Yaskawa INFORM job: ARGAZ_PROGRAM.JBI

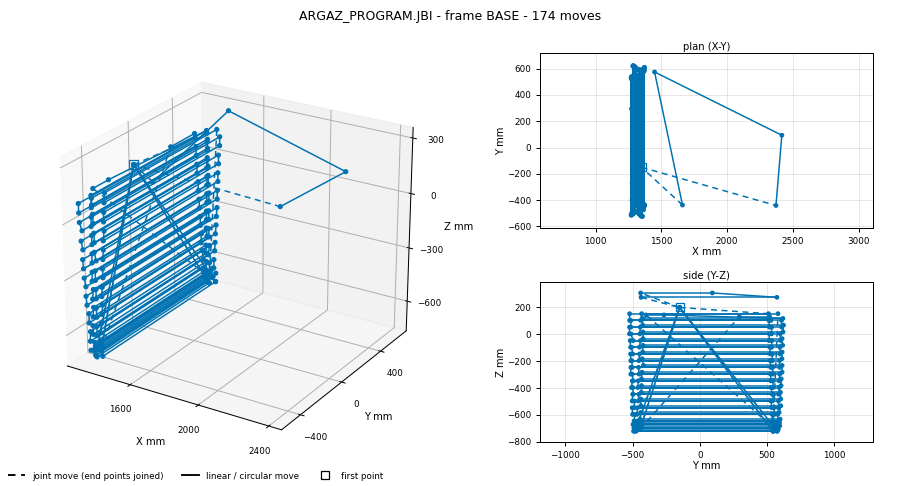
[picture p0: tool path of ARGAZ_PROGRAM.JBI in frame BASE, 174 of 174 moves have a stored position in this frame; points joined in program order, loops and branches not executed]
/JOB
//NAME ARGAZ_PROGRAM
//POS
///NPOS 168,0,168,1,0,1
///TOOL 0
///POSTYPE BASE
///RECTAN
///RCONF 0,0,0,0,0,0,0,0,0,0,0,0,0,0,0,0,0,0,0,0,0,0,0,0
C00000=2371.989,-440.401,308.020,175.0000,5.0000,90.0000
C00001=2416.705,93.738,308.020,175.0000,5.0000,90.0000
C00002=1448.862,574.607,275.381,175.0000,5.0000,90.0000
C00003=1661.240,-437.144,275.381,175.0000,5.0000,90.0000
C00004=1357.088,511.287,153.366,175.0000,-89.9999,5.0000
C00005=1357.088,-522.394,153.366,175.0000,-89.9999,5.0000
C00006=1354.164,-522.287,103.366,175.0000,-89.9999,5.0000
C00007=1354.164,514.938,103.366,175.0000,-89.9999,5.0000
C00008=1352.438,518.625,53.366,175.0000,-89.9999,5.0000
C00009=1352.438,-522.994,53.366,175.0000,-89.9999,5.0000
C00010=1350.832,-523.178,3.366,175.0000,-89.9999,5.0000
C00011=1350.832,518.871,3.366,175.0000,-89.9999,5.0000
C00012=1348.825,516.219,-46.633,175.0000,-89.9999,5.0000
C00013=1348.825,-518.107,-46.633,175.0000,-89.9999,5.0000
C00014=1347.044,-514.870,-96.633,175.0000,-89.9999,5.0000
C00015=1347.044,522.164,-96.633,175.0000,-89.9999,5.0000
C00016=1345.183,525.111,-146.633,175.0000,-89.9999,5.0000
C00017=1345.183,-515.018,-146.633,175.0000,-89.9999,5.0000
C00018=1343.293,-513.493,-196.633,175.0000,-89.9999,5.0000
C00019=1343.293,525.184,-196.633,175.0000,-89.9999,5.0000
C00020=1341.807,528.689,-246.633,175.0000,-89.9999,5.0000
C00021=1341.807,-512.923,-246.633,175.0000,-89.9999,5.0000
C00022=1339.870,-513.256,-296.633,175.0000,-89.9999,5.0000
C00023=1339.870,527.209,-296.633,175.0000,-89.9999,5.0000
C00024=1337.995,529.873,-346.633,175.0000,-89.9999,5.0000
C00025=1337.995,-502.334,-346.633,175.0000,-89.9999,5.0000
C00026=1336.213,-508.248,-396.633,175.0000,-89.9999,5.0000
C00027=1336.213,530.626,-396.633,175.0000,-89.9999,5.0000
C00028=1334.396,540.131,-446.633,175.0000,-89.9999,5.0000
C00029=1334.396,-499.231,-446.633,175.0000,-89.9999,5.0000
C00030=1332.129,-503.451,-496.633,175.0000,-89.9999,5.0000
C00031=1332.129,530.722,-496.633,175.0000,-89.9999,5.0000
C00032=1330.170,536.350,-546.633,175.0000,-89.9999,5.0000
C00033=1330.170,-503.270,-546.633,175.0000,-89.9999,5.0000
C00034=1328.250,-500.170,-596.633,175.0000,-89.9999,5.0000
C00035=1328.250,538.973,-596.633,175.0000,-89.9999,5.0000
C00036=1326.642,540.301,-646.633,175.0000,-89.9999,5.0000
C00037=1326.642,-487.964,-646.633,175.0000,-89.9999,5.0000
C00038=1324.806,-489.352,-696.633,175.0000,-89.9999,5.0000
C00039=1324.806,541.085,-696.633,175.0000,-89.9999,5.0000
C00040=1343.412,545.195,-671.633,180.0000,-60.0000,0.0000
C00041=1343.412,-497.251,-671.633,180.0000,-60.0000,0.0000
C00042=1342.156,-493.079,-721.633,180.0000,-60.0000,0.0000
C00043=1342.156,545.345,-721.633,180.0000,-60.0000,0.0000
C00044=1342.156,545.345,-721.633,180.0000,-60.0000,0.0000
C00045=1371.377,582.641,153.649,175.0000,-89.9999,5.0000
C00046=1371.377,-432.613,153.649,175.0000,-89.9999,5.0000
C00047=1372.180,-440.408,103.649,175.0000,-89.9999,5.0000
C00048=1372.180,609.123,103.649,175.0000,-89.9999,5.0000
C00049=1371.089,609.796,53.649,175.0000,-89.9999,5.0000
C00050=1371.089,-443.667,53.649,175.0000,-89.9999,5.0000
C00051=1369.998,-445.573,3.649,175.0000,-89.9999,5.0000
C00052=1369.998,599.394,3.649,175.0000,-89.9999,5.0000
C00053=1369.110,601.830,-46.350,175.0000,-89.9999,5.0000
C00054=1369.110,-441.873,-46.350,175.0000,-89.9999,5.0000
C00055=1367.639,-448.976,-96.350,175.0000,-89.9999,5.0000
C00056=1367.639,596.630,-96.350,175.0000,-89.9999,5.0000
C00057=1366.582,598.500,-146.350,175.0000,-89.9999,5.0000
C00058=1366.582,-448.746,-146.350,175.0000,-89.9999,5.0000
C00059=1365.085,-453.213,-196.350,175.0000,-89.9999,5.0000
C00060=1365.085,594.650,-196.350,175.0000,-89.9999,5.0000
C00061=1363.658,594.990,-246.350,175.0000,-89.9999,5.0000
C00062=1363.658,-455.754,-246.350,175.0000,-89.9999,5.0000
C00063=1361.864,-451.909,-296.350,175.0000,-89.9999,5.0000
C00064=1361.864,595.571,-296.350,175.0000,-89.9999,5.0000
C00065=1360.073,591.872,-346.350,175.0000,-89.9999,5.0000
C00066=1360.073,-458.655,-346.350,175.0000,-89.9999,5.0000
C00067=1358.161,-460.748,-396.350,175.0000,-89.9999,5.0000
C00068=1358.161,591.928,-396.350,175.0000,-89.9999,5.0000
C00069=1356.405,587.009,-446.350,175.0000,-89.9999,5.0000
C00070=1356.405,-453.709,-446.350,175.0000,-89.9999,5.0000
C00071=1354.608,-458.341,-496.350,175.0000,-89.9999,5.0000
C00072=1354.608,586.376,-496.350,175.0000,-89.9999,5.0000
C00073=1352.468,585.807,-546.350,175.0000,-89.9999,5.0000
C00074=1352.468,-463.981,-546.350,175.0000,-89.9999,5.0000
C00075=1350.405,-467.600,-596.350,175.0000,-89.9999,5.0000
C00076=1350.405,580.519,-596.350,175.0000,-89.9999,5.0000
C00077=1348.479,582.258,-646.350,175.0000,-89.9999,5.0000
C00078=1348.479,-467.412,-646.350,175.0000,-89.9999,5.0000
C00079=1346.462,-469.588,-696.350,175.0000,-89.9999,5.0000
C00080=1346.462,577.739,-696.350,175.0000,-89.9999,5.0000
C00081=1364.869,576.218,-671.350,180.0000,-60.0000,0.0000
C00082=1364.869,-472.867,-671.350,180.0000,-60.0000,0.0000
C00083=1363.104,-472.908,-721.350,180.0000,-60.0000,0.0000
C00084=1363.104,576.344,-721.350,180.0000,-60.0000,0.0000
C00085=1363.104,576.344,-721.350,180.0000,-60.0000,0.0000
C00086=1277.888,-399.618,144.199,175.0000,-89.9999,5.0000
C00087=1277.888,-266.558,144.199,175.0000,-89.9999,5.0000
C00088=1283.410,619.398,117.816,175.0000,-89.9999,5.0000
C00089=1283.410,-424.812,117.816,175.0000,-89.9999,5.0000
C00090=1286.253,-425.480,67.816,175.0000,-89.9999,5.0000
C00091=1286.253,623.737,67.816,175.0000,-89.9999,5.0000
C00092=1288.733,620.101,17.816,175.0000,-89.9999,5.0000
C00093=1288.733,-423.231,17.816,175.0000,-89.9999,5.0000
C00094=1291.050,-422.345,-32.183,175.0000,-89.9999,5.0000
C00095=1291.050,613.233,-32.183,175.0000,-89.9999,5.0000
C00096=1293.592,617.319,-82.183,175.0000,-89.9999,5.0000
C00097=1293.592,-423.386,-82.183,175.0000,-89.9999,5.0000
C00098=1295.614,-424.881,-132.183,175.0000,-89.9999,5.0000
C00099=1295.614,613.520,-132.183,175.0000,-89.9999,5.0000
C00100=1297.247,612.008,-182.183,175.0000,-89.9999,5.0000
C00101=1297.247,-429.228,-182.183,175.0000,-89.9999,5.0000
C00102=1299.433,-419.216,-232.183,175.0000,-89.9999,5.0000
C00103=1299.433,613.471,-232.183,175.0000,-89.9999,5.0000
C00104=1300.418,613.420,-282.183,175.0000,-89.9999,5.0000
C00105=1300.418,-430.256,-282.183,175.0000,-89.9999,5.0000
C00106=1302.234,-433.734,-332.183,175.0000,-89.9999,5.0000
C00107=1302.234,606.925,-332.183,175.0000,-89.9999,5.0000
C00108=1303.707,605.868,-382.183,175.0000,-89.9999,5.0000
C00109=1303.707,-433.869,-382.183,175.0000,-89.9999,5.0000
C00110=1305.086,-435.019,-432.183,175.0000,-89.9999,5.0000
C00111=1305.086,600.756,-432.183,175.0000,-89.9999,5.0000
C00112=1306.071,603.429,-482.183,175.0000,-89.9999,5.0000
C00113=1306.071,-438.802,-482.183,175.0000,-89.9999,5.0000
C00114=1307.412,-438.117,-532.183,175.0000,-89.9999,5.0000
C00115=1307.412,603.875,-532.183,175.0000,-89.9999,5.0000
C00116=1308.466,591.089,-582.183,175.0000,-89.9999,5.0000
C00117=1308.466,-439.996,-582.183,175.0000,-89.9999,5.0000
C00118=1310.304,-445.204,-632.183,175.0000,-89.9999,5.0000
C00119=1310.304,598.888,-632.183,175.0000,-89.9999,5.0000
C00120=1311.312,595.813,-682.183,175.0000,-89.9999,5.0000
C00121=1311.312,-443.494,-682.183,175.0000,-89.9999,5.0000
C00122=1332.658,-435.818,-657.183,180.0000,-60.0000,0.0000
C00123=1332.658,594.168,-657.183,180.0000,-60.0000,0.0000
C00124=1333.118,585.110,-707.183,180.0000,-60.0000,0.0000
C00125=1333.118,-444.618,-707.183,180.0000,-60.0000,0.0000
C00126=1333.118,-444.618,-707.183,180.0000,-60.0000,0.0000
C00127=1273.288,295.502,131.277,175.0000,-89.9999,5.0000
C00128=1273.288,520.035,131.277,175.0000,-89.9999,5.0000
C00129=1270.890,529.755,103.296,175.0000,-89.9999,5.0000
C00130=1270.890,-513.266,103.296,175.0000,-89.9999,5.0000
C00131=1271.533,-513.209,53.296,175.0000,-89.9999,5.0000
C00132=1271.533,535.502,53.296,175.0000,-89.9999,5.0000
C00133=1273.366,534.257,3.296,175.0000,-89.9999,5.0000
C00134=1273.366,-513.096,3.296,175.0000,-89.9999,5.0000
C00135=1275.404,-495.948,-46.703,175.0000,-89.9999,5.0000
C00136=1275.404,536.502,-46.703,175.0000,-89.9999,5.0000
C00137=1277.028,534.815,-96.703,175.0000,-89.9999,5.0000
C00138=1277.028,-508.386,-96.703,175.0000,-89.9999,5.0000
C00139=1279.183,-498.977,-146.703,175.0000,-89.9999,5.0000
C00140=1279.183,540.662,-146.703,175.0000,-89.9999,5.0000
C00141=1280.966,539.787,-196.703,175.0000,-89.9999,5.0000
C00142=1280.966,-505.503,-196.703,175.0000,-89.9999,5.0000
C00143=1282.925,-503.396,-246.703,175.0000,-89.9999,5.0000
C00144=1282.925,542.645,-246.703,175.0000,-89.9999,5.0000
C00145=1285.047,543.565,-296.703,175.0000,-89.9999,5.0000
C00146=1285.047,-503.499,-296.703,175.0000,-89.9999,5.0000
C00147=1287.369,-494.427,-346.703,175.0000,-89.9999,5.0000
C00148=1287.369,546.345,-346.703,175.0000,-89.9999,5.0000
C00149=1289.521,543.757,-396.703,175.0000,-89.9999,5.0000
C00150=1289.521,-498.930,-396.703,175.0000,-89.9999,5.0000
C00151=1291.635,-495.764,-446.703,175.0000,-89.9999,5.0000
C00152=1291.635,549.175,-446.703,175.0000,-89.9999,5.0000
C00153=1293.849,541.736,-496.703,175.0000,-89.9999,5.0000
C00154=1293.849,-485.793,-496.703,175.0000,-89.9999,5.0000
C00155=1295.977,-487.912,-546.703,175.0000,-89.9999,5.0000
C00156=1295.977,552.744,-546.703,175.0000,-89.9999,5.0000
C00157=1298.303,555.349,-596.703,175.0000,-89.9999,5.0000
C00158=1298.303,-482.618,-596.703,175.0000,-89.9999,5.0000
C00159=1300.270,-489.107,-646.703,175.0000,-89.9999,5.0000
C00160=1300.270,549.567,-646.703,175.0000,-89.9999,5.0000
C00161=1302.656,551.655,-696.703,175.0000,-89.9999,5.0000
C00162=1302.656,-488.761,-696.703,175.0000,-89.9999,5.0000
C00163=1324.870,-481.376,-671.703,180.0000,-60.0000,0.0000
C00164=1324.870,551.349,-671.703,180.0000,-60.0000,0.0000
C00165=1327.105,551.261,-721.703,180.0000,-60.0000,0.0000
C00166=1327.105,-481.969,-721.703,180.0000,-60.0000,0.0000
C00167=1327.105,-481.969,-721.703,180.0000,-60.0000,0.0000
///POSTYPE PULSE
///PULSE
EC00000=0
EC00001=0
EC00002=0
EC00003=0
EC00004=0
EC00005=0
EC00006=0
EC00007=0
EC00008=0
EC00009=0
EC00010=0
EC00011=0
EC00012=0
EC00013=0
EC00014=0
EC00015=0
EC00016=0
EC00017=0
EC00018=0
EC00019=0
EC00020=0
EC00021=0
EC00022=0
EC00023=0
EC00024=0
EC00025=0
EC00026=0
EC00027=0
EC00028=0
EC00029=0
EC00030=0
EC00031=0
EC00032=0
EC00033=0
EC00034=0
EC00035=0
EC00036=0
EC00037=0
EC00038=0
EC00039=0
EC00040=0
EC00041=0
EC00042=0
EC00043=0
EC00044=92160
EC00045=92160
EC00046=92160
EC00047=92160
EC00048=92160
EC00049=92160
EC00050=92160
EC00051=92160
EC00052=92160
EC00053=92160
EC00054=92160
EC00055=92160
EC00056=92160
EC00057=92160
EC00058=92160
EC00059=92160
EC00060=92160
EC00061=92160
EC00062=92160
EC00063=92160
EC00064=92160
EC00065=92160
EC00066=92160
EC00067=92160
EC00068=92160
EC00069=92160
EC00070=92160
EC00071=92160
EC00072=92160
EC00073=92160
EC00074=92160
EC00075=92160
EC00076=92160
EC00077=92160
EC00078=92160
EC00079=92160
EC00080=92160
EC00081=92160
EC00082=92160
EC00083=92160
EC00084=92160
EC00085=184320
EC00086=184320
EC00087=184320
EC00088=184320
EC00089=184320
EC00090=184320
EC00091=184320
EC00092=184320
EC00093=184320
EC00094=184320
EC00095=184320
EC00096=184320
EC00097=184320
EC00098=184320
EC00099=184320
EC00100=184320
EC00101=184320
EC00102=184320
EC00103=184320
EC00104=184320
EC00105=184320
EC00106=184320
EC00107=184320
EC00108=184320
EC00109=184320
EC00110=184320
EC00111=184320
EC00112=184320
EC00113=184320
EC00114=184320
EC00115=184320
EC00116=184320
EC00117=184320
EC00118=184320
EC00119=184320
EC00120=184320
EC00121=184320
EC00122=184320
EC00123=184320
EC00124=184320
EC00125=184320
EC00126=276480
EC00127=276480
EC00128=276480
EC00129=276480
EC00130=276480
EC00131=276480
EC00132=276480
EC00133=276480
EC00134=276480
EC00135=276480
EC00136=276480
EC00137=276480
EC00138=276480
EC00139=276480
EC00140=276480
EC00141=276480
EC00142=276480
EC00143=276480
EC00144=276480
EC00145=276480
EC00146=276480
EC00147=276480
EC00148=276480
EC00149=276480
EC00150=276480
EC00151=276480
EC00152=276480
EC00153=276480
EC00154=276480
EC00155=276480
EC00156=276480
EC00157=276480
EC00158=276480
EC00159=276480
EC00160=276480
EC00161=276480
EC00162=276480
EC00163=276480
EC00164=276480
EC00165=276480
EC00166=276480
EC00167=368640
///POSTYPE BASE
///RECTAN
///RCONF 1,0,0,0,0,0,0,0,0,0,0,0,0,0,0,0,0,0,0,0,0,0,0,0
P00009=1350.000,-150.000,200.000,-180.0000,-45.0000,0.0000
///POSTYPE PULSE
///PULSE
EX00000=0
//INST
///DATE 2023/01/29 12:01
///ATTR SC,RW,RJ
////FRAME BASE
///GROUP1 RB1,ST1
NOP
MOVJ P009 EX000 VJ=15.00
MOVJ C00000 EC00000 VJ=15.00
CALL JOB:SPYON
MOVL C00001 EC00001 V=150.0
MOVL C00002 EC00002 V=150.0
MOVL C00003 EC00003 V=150.0
CALL JOB:SPYOF
MOVJ P009 VJ=15.00
MOVJ C00004 EC00004 VJ=15.00
CALL JOB:SPYON
MOVL C00005 EC00005 V=150.0
MOVL C00006 EC00006 V=150.0
MOVL C00007 EC00007 V=150.0
MOVL C00008 EC00008 V=150.0
MOVL C00009 EC00009 V=150.0
MOVL C00010 EC00010 V=150.0
MOVL C00011 EC00011 V=150.0
MOVL C00012 EC00012 V=150.0
MOVL C00013 EC00013 V=150.0
MOVL C00014 EC00014 V=150.0
MOVL C00015 EC00015 V=150.0
MOVL C00016 EC00016 V=150.0
MOVL C00017 EC00017 V=150.0
MOVL C00018 EC00018 V=150.0
MOVL C00019 EC00019 V=150.0
MOVL C00020 EC00020 V=150.0
MOVL C00021 EC00021 V=150.0
MOVL C00022 EC00022 V=150.0
MOVL C00023 EC00023 V=150.0
MOVL C00024 EC00024 V=150.0
MOVL C00025 EC00025 V=150.0
MOVL C00026 EC00026 V=150.0
MOVL C00027 EC00027 V=150.0
MOVL C00028 EC00028 V=150.0
MOVL C00029 EC00029 V=150.0
MOVL C00030 EC00030 V=150.0
MOVL C00031 EC00031 V=150.0
MOVL C00032 EC00032 V=150.0
MOVL C00033 EC00033 V=150.0
MOVL C00034 EC00034 V=150.0
MOVL C00035 EC00035 V=150.0
MOVL C00036 EC00036 V=150.0
MOVL C00037 EC00037 V=150.0
MOVL C00038 EC00038 V=150.0
MOVL C00039 EC00039 V=150.0
MOVL C00040 EC00040 V=150.0
MOVL C00041 EC00041 V=150.0
MOVL C00042 EC00042 V=150.0
MOVL C00043 EC00043 V=150.0
CALL JOB:SPYOF
MOVJ P009 VJ=15.00
MOVL C00044 EC00044 V=150.0
MOVJ C00045 EC00045 VJ=15.00
CALL JOB:SPYON
MOVL C00046 EC00046 V=150.0
MOVL C00047 EC00047 V=150.0
MOVL C00048 EC00048 V=150.0
MOVL C00049 EC00049 V=150.0
MOVL C00050 EC00050 V=150.0
MOVL C00051 EC00051 V=150.0
MOVL C00052 EC00052 V=150.0
MOVL C00053 EC00053 V=150.0
MOVL C00054 EC00054 V=150.0
MOVL C00055 EC00055 V=150.0
MOVL C00056 EC00056 V=150.0
MOVL C00057 EC00057 V=150.0
MOVL C00058 EC00058 V=150.0
MOVL C00059 EC00059 V=150.0
MOVL C00060 EC00060 V=150.0
MOVL C00061 EC00061 V=150.0
MOVL C00062 EC00062 V=150.0
MOVL C00063 EC00063 V=150.0
MOVL C00064 EC00064 V=150.0
MOVL C00065 EC00065 V=150.0
MOVL C00066 EC00066 V=150.0
MOVL C00067 EC00067 V=150.0
MOVL C00068 EC00068 V=150.0
MOVL C00069 EC00069 V=150.0
MOVL C00070 EC00070 V=150.0
MOVL C00071 EC00071 V=150.0
MOVL C00072 EC00072 V=150.0
MOVL C00073 EC00073 V=150.0
MOVL C00074 EC00074 V=150.0
MOVL C00075 EC00075 V=150.0
MOVL C00076 EC00076 V=150.0
MOVL C00077 EC00077 V=150.0
MOVL C00078 EC00078 V=150.0
MOVL C00079 EC00079 V=150.0
MOVL C00080 EC00080 V=150.0
MOVL C00081 EC00081 V=150.0
MOVL C00082 EC00082 V=150.0
MOVL C00083 EC00083 V=150.0
MOVL C00084 EC00084 V=150.0
CALL JOB:SPYOF
MOVJ P009 VJ=15.00
MOVL C00085 EC00085 V=150.0
MOVJ C00086 EC00086 VJ=15.00
CALL JOB:SPYON
MOVL C00087 EC00087 V=150.0
MOVL C00088 EC00088 V=150.0
MOVL C00089 EC00089 V=150.0
MOVL C00090 EC00090 V=150.0
MOVL C00091 EC00091 V=150.0
MOVL C00092 EC00092 V=150.0
MOVL C00093 EC00093 V=150.0
MOVL C00094 EC00094 V=150.0
MOVL C00095 EC00095 V=150.0
MOVL C00096 EC00096 V=150.0
MOVL C00097 EC00097 V=150.0
MOVL C00098 EC00098 V=150.0
MOVL C00099 EC00099 V=150.0
MOVL C00100 EC00100 V=150.0
MOVL C00101 EC00101 V=150.0
MOVL C00102 EC00102 V=150.0
MOVL C00103 EC00103 V=150.0
MOVL C00104 EC00104 V=150.0
MOVL C00105 EC00105 V=150.0
MOVL C00106 EC00106 V=150.0
MOVL C00107 EC00107 V=150.0
MOVL C00108 EC00108 V=150.0
MOVL C00109 EC00109 V=150.0
MOVL C00110 EC00110 V=150.0
MOVL C00111 EC00111 V=150.0
MOVL C00112 EC00112 V=150.0
MOVL C00113 EC00113 V=150.0
MOVL C00114 EC00114 V=150.0
MOVL C00115 EC00115 V=150.0
MOVL C00116 EC00116 V=150.0
MOVL C00117 EC00117 V=150.0
MOVL C00118 EC00118 V=150.0
MOVL C00119 EC00119 V=150.0
MOVL C00120 EC00120 V=150.0
MOVL C00121 EC00121 V=150.0
MOVL C00122 EC00122 V=150.0
MOVL C00123 EC00123 V=150.0
MOVL C00124 EC00124 V=150.0
MOVL C00125 EC00125 V=150.0
CALL JOB:SPYOF
MOVJ P009 VJ=15.00
MOVL C00126 EC00126 V=150.0
MOVJ C00127 EC00127 VJ=15.00
CALL JOB:SPYON
MOVL C00128 EC00128 V=150.0
MOVL C00129 EC00129 V=150.0
MOVL C00130 EC00130 V=150.0
MOVL C00131 EC00131 V=150.0
MOVL C00132 EC00132 V=150.0
MOVL C00133 EC00133 V=150.0
MOVL C00134 EC00134 V=150.0
MOVL C00135 EC00135 V=150.0
MOVL C00136 EC00136 V=150.0
MOVL C00137 EC00137 V=150.0
MOVL C00138 EC00138 V=150.0
MOVL C00139 EC00139 V=150.0
MOVL C00140 EC00140 V=150.0
MOVL C00141 EC00141 V=150.0
MOVL C00142 EC00142 V=150.0
MOVL C00143 EC00143 V=150.0
MOVL C00144 EC00144 V=150.0
MOVL C00145 EC00145 V=150.0
MOVL C00146 EC00146 V=150.0
MOVL C00147 EC00147 V=150.0
MOVL C00148 EC00148 V=150.0
MOVL C00149 EC00149 V=150.0
MOVL C00150 EC00150 V=150.0
MOVL C00151 EC00151 V=150.0
MOVL C00152 EC00152 V=150.0
MOVL C00153 EC00153 V=150.0
MOVL C00154 EC00154 V=150.0
MOVL C00155 EC00155 V=150.0
MOVL C00156 EC00156 V=150.0
MOVL C00157 EC00157 V=150.0
MOVL C00158 EC00158 V=150.0
MOVL C00159 EC00159 V=150.0
MOVL C00160 EC00160 V=150.0
MOVL C00161 EC00161 V=150.0
MOVL C00162 EC00162 V=150.0
MOVL C00163 EC00163 V=150.0
MOVL C00164 EC00164 V=150.0
MOVL C00165 EC00165 V=150.0
MOVL C00166 EC00166 V=150.0
CALL JOB:SPYOF
MOVJ P009 VJ=15.00
MOVL C00167 EC00167 V=150.0
END
